(* PLC project faults, TNI-Software ControlBuild 4.00.18 *)
(* stored: creationDateTime 2005-06-22T10:04:43-01:00 *)

FUNCTION_BLOCK batch.faults
  VAR_INPUT  (* CB.kind=inputVars *)
    generalFault1 : BOOL := false;  (* CB.mnemonicPatternPropertyName=defGeneral<SY><NU> CB.libelle=Défaut général *)
    generalFault2 : BOOL := false;  (* CB.mnemonicPatternPropertyName=defGeneral<SY><NU> CB.libelle=Défaut général *)
    generalFault3 : BOOL := false;  (* CB.mnemonicPatternPropertyName=defGeneral<SY><NU> CB.libelle=Défaut général *)
    generalFault4 : BOOL := false;  (* CB.mnemonicPatternPropertyName=defGeneral<SY><NU> CB.libelle=Défaut général *)
  END_VAR
  VAR_OUTPUT  (* CB.kind=outputVars *)
    fault : BOOL := false;  (* CB.mnemonicPatternPropertyName=fault<SY><NU> *)
  END_VAR

(* LD diagram, written out as Structured Text *)
1:
fault := generalFault4 OR generalFault1 OR generalFault2 OR generalFault3;
END_FUNCTION_BLOCK
